(* 
## Short summary

This class is a data transfer object for configurable cycle time recorder attributes. 
It is intended to be uses within a fluid configuration interface. 

.. <legal notes>

legal notes
=================
| SPDX-FileCopyrightText: © 2025 ekvip automation GmbH <info@ekvip.de>
| SPDX-License-Identifier: Apache-2.0
| For details check: Apache-2.0_

.. _Apache-2.0: https://www.apache.org/licenses/LICENSE-2.0

.. </legal notes>

*)

FUNCTION_BLOCK CycleTimeRecorderConfiguration EXTENDS DefaultMeasurementConfiguration IMPLEMENTS CNM_ProductionMetricInterfaces.ICycleTimeConfiguration
VAR
	configuredTargetCycleTime :LTIME;
END_VAR

(*

## Short summary

This abstract property returns the class name of the concrete object, 
which is useful for logging/debugging purpose or to check the class name
for ``__DELETE`` in factories (sometimes it's necessary to do more 
than just to free the memory).

.. <legal notes>

legal notes
=================
| SPDX-FileCopyrightText: © 2022 ekvip automation GmbH <info@ekvip.de>
| SPDX-License-Identifier: Apache-2.0
| For details check: Apache-2.0_

.. _Apache-2.0: https://www.apache.org/licenses/LICENSE-2.0

.. </legal notes>

*)
PROPERTY className : CNM_AbstractObject.ClassName
GET
className := 'CycleTimeRecorderConfiguration';
END_GET
END_PROPERTY

(* 
## Short summary

This property can be used to set and read the current target cycle time for a product cycle of a single part.
The target cycle time will be written into every measurement entry and is used to mark cycle time exceedances.

.. <legal notes>

legal notes
=================
| SPDX-FileCopyrightText: © 2025 ekvip automation GmbH <info@ekvip.de>
| SPDX-License-Identifier: Apache-2.0
| For details check: Apache-2.0_

.. _Apache-2.0: https://www.apache.org/licenses/LICENSE-2.0

.. </legal notes>

*)
PROPERTY targetCycleTime : LTIME
GET
targetCycleTime := THIS^.configuredTargetCycleTime;
END_GET
SET
THIS^.configuredTargetCycleTime := targetCycleTime;
END_SET
END_PROPERTY

END_FUNCTION_BLOCK

(* stored: Version 1.1.0.1
   POU CycleTimeRecorderConfiguration: Id {e53a104d-d70c-46aa-9137-d54b33709f10}, SpecialFunc None
   Property className: Id {5b3c2050-1491-4137-813d-69099ec07532}
   Get Get: Id {db212f4d-fd9a-49fe-add5-92f72a479960}
   Property targetCycleTime: Id {00ba80c0-ada5-427e-96a3-9bdb8c351a97}
   Get Get: Id {4e8a7b3f-7676-4747-9d94-094f61a93fba}
   Set Set: Id {a4f0cf7e-2142-4a26-a365-27c7ece0a749} *)
